FUNCTION_BLOCK StructuredDatatype_TestSuite EXTENDS TcUnit.FB_TestSuite
VAR
END_VAR

TestAddress();
TestClearReference();
TestClone();
TestTypeNameReturnsExpected();
TestIdentifierReturnsExpected();
TestMakeReferenceToFollowsReference();
TestMakeReferenceToUpdatesReference();
TestSize();
TestValueReturnsExpectedAfterChange();
TestSerializeTypeWith();
TestSerializeWith();
TestTryDeserializeFrom();
TestTryMakeReferenceToFollowsReference();
TestTryMakeReferenceToUpdatesReference();

METHOD PUBLIC TestAddress
VAR
    _type : MockStructuredDatatype_TIMESTRUCT;
    notExpected : PVOID := 0;
    actual : PVOID;
END_VAR
TEST('TestAddress');

actual := _type.Address;

AssertFalse(
    Condition := (notExpected = actual),
    Message := 'Type did not return a valid address.'
);

TEST_FINISHED();
END_METHOD

METHOD PUBLIC TestClearReference
VAR
    _type : MockStructuredDatatype_TIMESTRUCT;
	target : TIMESTRUCT;
    expected : TIMESTRUCT;
    actual : TIMESTRUCT;
END_VAR
TEST('TestClearReference');

_type.MakeReferenceTo(target);
_type.ClearReference();
target.wDay := 2;

actual := _type.Value;

AssertEquals(
    Expected := expected,
    Actual := actual,
    Message := 'Value incorrectly followed target change'
);

TEST_FINISHED();
END_METHOD

METHOD PUBLIC TestClone
VAR
    _type : MockStructuredDatatype_TIMESTRUCT;
	clone : I_Datatype;
	isValidClone : BOOL;
	compareResult : DINT;
END_VAR
TEST('TestClone');

clone := _type.Clone();

isValidClone := clone <> 0;

IF isValidClone THEN
	compareResult := memcmp(_type.Address, clone.Address, clone.Size);
END_IF

AssertTrue(
	Condition := isValidClone,
	Message := 'Clone did not produce a clone'
);

AssertEquals_DINT(
	Expected := 0,
    Actual := compareResult,
    Message := 'Clone did not return a valid clone.'
);

clone.Dispose();

TEST_FINISHED();
END_METHOD

METHOD PUBLIC TestIdentifierReturnsExpected
VAR
    _type : MockStructuredDatatype_TIMESTRUCT;
    expected : STRING := 'TIMESTRUCT';
    actual : STRING;
END_VAR
TEST('TestIdentifierReturnsExpected');

actual := _type.Identifier;

AssertEquals_STRING(
    Expected := expected,
    Actual := actual,
    Message := 'Type did not return correct iec type.'
);

TEST_FINISHED();
END_METHOD

METHOD PUBLIC TestMakeReferenceToFollowsReference
VAR
    _type : MockStructuredDatatype_TIMESTRUCT;
	target : TIMESTRUCT;
    expected : TIMESTRUCT := (wDay := 2);
    actual : TIMESTRUCT;
END_VAR
TEST('TestMakeReferenceToFollowsReference');

_type.MakeReferenceTo(target);
target.wDay := 2;

actual := _type.Value;

AssertEquals(
    Expected := expected,
    Actual := actual,
    Message := 'Value did not follow target change'
);

TEST_FINISHED();
END_METHOD

METHOD PUBLIC TestMakeReferenceToUpdatesReference
VAR
    _type : MockStructuredDatatype_TIMESTRUCT;
	target : TIMESTRUCT;
    expected : TIMESTRUCT := (wDay := 2);
    actual : TIMESTRUCT;
END_VAR
TEST('TestMakeReferenceToUpdatesReference');

_type.MakeReferenceTo(target);
_type.wDay.Value := 2;

actual := target;

AssertEquals(
    Expected := expected,
    Actual := actual,
    Message := 'Value did not update target'
);

TEST_FINISHED();
END_METHOD

METHOD PUBLIC TestSerializeTypeWith
VAR
    _type : MockStructuredDatatype_TIMESTRUCT;
    serializer : JsonSerializer;
    expected : STRING(1000) := '{"typeName":"STRUCT","identifier":"TIMESTRUCT","members":{"wYear":{"typeName":"WORD","minValue":0,"maxValue":65535,"isSigned":false,"isFloat":false},"wMonth":{"typeName":"WORD","minValue":0,"maxValue":65535,"isSigned":false,"isFloat":false},"wDayOfWeek":{"typeName":"WORD","minValue":0,"maxValue":65535,"isSigned":false,"isFloat":false},"wDay":{"typeName":"WORD","minValue":0,"maxValue":65535,"isSigned":false,"isFloat":false},"wHour":{"typeName":"WORD","minValue":0,"maxValue":65535,"isSigned":false,"isFloat":false},"wMinute":{"typeName":"WORD","minValue":0,"maxValue":65535,"isSigned":false,"isFloat":false},"wSecond":{"typeName":"WORD","minValue":0,"maxValue":65535,"isSigned":false,"isFloat":false},"wMilliseconds":{"typeName":"WORD","minValue":0,"maxValue":65535,"isSigned":false,"isFloat":false}}}';
    actual : STRING(1000);
END_VAR
TEST('TestSerializeTypeWith');

serializer.Reset();
_type.SerializeTypeWith(serializer);
serializer.TryGetSerializedData(ADR(actual), SIZEOF(actual));

AssertEquals_STRING(
    Expected := expected,
    Actual := actual,
    Message := 'Serialization of type did not return correct string.'
);

TEST_FINISHED();
END_METHOD

METHOD PUBLIC TestSerializeWith
VAR
    _type : MockStructuredDatatype_TIMESTRUCT;
    serializer : JsonSerializer;
    expected : STRING(500) := '{"wYear":2000,"wMonth":1,"wDayOfWeek":2,"wDay":3,"wHour":4,"wMinute":5,"wSecond":6,"wMilliseconds":7}';
    actual : STRING(500);
END_VAR
TEST('TestSerializeWith');

_type.wYear.Value := 2000;
_type.wMonth.Value := 1;
_type.wDayOfWeek.Value := 2;
_type.wDay.Value := 3;
_type.wHour.Value := 4;
_type.wMinute.Value := 5;
_type.wSecond.Value := 6;
_type.wMilliseconds.Value := 7;

serializer.Reset();
_type.SerializeWith(serializer);
serializer.TryGetSerializedData(ADR(actual), SIZEOF(actual));

AssertEquals_STRING(
    Expected := expected,
    Actual := actual,
    Message := 'Serialization of type data did not return correct string.'
);

TEST_FINISHED();
END_METHOD

METHOD PUBLIC TestSize
VAR
    _type : MockStructuredDatatype_TIMESTRUCT;
    expected : UDINT := SIZEOF(TIMESTRUCT);
    actual : UDINT;
END_VAR
TEST('TestSize');

actual := _type.Size;

AssertEquals_UDINT(
    Expected := Expected,
    Actual := actual,
    Message := 'Type did not return the correct size.'
);

TEST_FINISHED();
END_METHOD

METHOD PUBLIC TestTryDeserializeFrom
VAR
    deserializer : JsonDeserializer;
    feedback : DeserializerFeedback;
    json : STRING(500) := '{"wDay":3,"wDayOfWeek":2,"wHour":4,"wMilliseconds":7,"wMinute":5,"wMonth":1,"wSecond":6,"wYear":2000}';
    _type : MockStructuredDatatype_TIMESTRUCT;
    expected : TIMESTRUCT := (wYear := 2000, wMonth := 1, wDayOfWeek := 2, wDay := 3, wHour := 4, wMinute := 5, wSecond := 6, wMilliseconds := 7);
    actual : TIMESTRUCT;
 END_VAR
TEST('TestTryDeserializeFrom');

deserializer.Reset();
deserializer.TryLoad(json);
_type.TryDeserializeFrom(Deserializer, Feedback);

actual := _type.Value;

AssertEquals(
    Expected := expected,
    Actual := actual,
    Message := 'Type did not deserialize correctly.'
);

TEST_FINISHED();
END_METHOD

METHOD PUBLIC TestTryMakeReferenceToFollowsReference
VAR
    _type : MockStructuredDatatype_TIMESTRUCT;
	target : MockStructuredDatatype_TIMESTRUCT;
    expected : TIMESTRUCT := (wDay := 2);
    actual : TIMESTRUCT;
END_VAR
TEST('TestTryMakeReferenceToFollowsReference');

_type.TryMakeReferenceTo(target);
target.wDay.Value := 2;

actual := _type.Value;

AssertEquals(
    Expected := expected,
    Actual := actual,
    Message := 'Value did not follow target change'
);

TEST_FINISHED();
END_METHOD

METHOD PUBLIC TestTryMakeReferenceToUpdatesReference
VAR
    _type : MockStructuredDatatype_TIMESTRUCT;
	target : MockStructuredDatatype_TIMESTRUCT;
    expected : TIMESTRUCT := (wDay := 2);
    actual : TIMESTRUCT;
END_VAR
TEST('TestTryMakeReferenceToUpdatesReference');

_type.TryMakeReferenceTo(target);
_type.wDay.Value := 2;

actual := target.Value;

AssertEquals(
    Expected := expected,
    Actual := actual,
    Message := 'Value did not update target'
);

TEST_FINISHED();
END_METHOD

METHOD PUBLIC TestTypeNameReturnsExpected
VAR
    _type : MockStructuredDatatype_TIMESTRUCT;
    expected : STRING := 'STRUCT';
    actual : STRING;
END_VAR
TEST('TestTypeNameReturnsExpected');

actual := _type.TypeName;

AssertEquals_STRING(
    Expected := expected,
    Actual := actual,
    Message := 'Type did not return correct iec type.'
);

TEST_FINISHED();
END_METHOD

METHOD PUBLIC TestValueReturnsExpectedAfterChange
VAR
    _type : MockStructuredDatatype_TIMESTRUCT;
	value : TIMESTRUCT := (wDay := 2);
    expected : TIMESTRUCT := (wDay := 2);
    actual : TIMESTRUCT;
END_VAR
TEST('TestValueReturnsExpectedAfterChange');

_type.Value := value;
actual := _type.Value;

AssertEquals(
    Expected := expected,
    Actual := actual,
    Message := 'Expected value not returned after change.'
);

TEST_FINISHED();
END_METHOD

END_FUNCTION_BLOCK

(* stored: Version 1.1.0.1, ProductVersion 3.1.4024.12
   POU StructuredDatatype_TestSuite: Id {8da4ed46-1d64-0989-004e-ca94ba643016}, SpecialFunc None
   Method TestAddress: Id {8d0a9c63-fba4-0aa0-1310-2e8d90ecb63c}
   Method TestClearReference: Id {41bee5eb-e0ac-09c8-178d-901dfdff62d7}
   Method TestClone: Id {bf7abec4-329a-0cac-256b-46d44242b42c}
   Method TestIdentifierReturnsExpected: Id {4638ddca-f28a-0bb3-2a52-1b4f82e9af01}
   Method TestMakeReferenceToFollowsReference: Id {cc2427de-9ee5-0fd7-1db0-f899702c2193}
   Method TestMakeReferenceToUpdatesReference: Id {ac141f91-f598-09bc-27cd-ac724f02c8ca}
   Method TestSerializeTypeWith: Id {ce7f2189-873b-082f-2b63-a9cc50488a68}
   Method TestSerializeWith: Id {af97f698-50fc-0d6e-39ca-5252997b0526}
   Method TestSize: Id {992c5f1e-6206-0965-2bd7-1ea550a96d06}
   Method TestTryDeserializeFrom: Id {1e40072b-f85e-0476-1596-611f654da5f5}
   Method TestTryMakeReferenceToFollowsReference: Id {74a2dd17-7c7a-01f4-23d6-f6f176926afa}
   Method TestTryMakeReferenceToUpdatesReference: Id {ceb54fd6-7dc2-0a8b-017b-2d4924bdaf62}
   Method TestTypeNameReturnsExpected: Id {4c61d39e-36cb-0beb-037c-8a84619a2a20}
   Method TestValueReturnsExpectedAfterChange: Id {ee0b88af-88a6-0b64-3957-3851d963ea7d} *)
